TYPE "PathTestHMI"
VERSION : 0.1
// Block: PathTestHMI
   STRUCT
      ManCmdStartTest : Bool;
      TestEnabled : Bool;
      TestRequired : Bool;
      TestStarted : Bool;
      TestRunning : Bool;
   END_STRUCT;

END_TYPE
